PROGRAM P61_AO
VAR
	//ACT_Ramp_OLD();
	MFC01, MFC02, MFC03, MFC04, MFC05, MFC06, MFC07, MFC08, MFC09, MFC10: FB_Ramp2;
	MFC11, MFC12, MFC13, MFC14, MFC15, MFC16, MFC17, MFC18, MFC19: FB_Ramp2;		
	EPC01, EPC02, EPC03, EPC04, EPC05, EPC06, EPC07: FB_Ramp2;	
	IH, ROT, POS, P01: FB_Ramp2;
		
	//HT01: FB_Ramp2;
	halfRes: REAL := 16383;//0~5V
	fullRes: REAL := 32767;//0~10V or 4~20mA
	halfRes_ROT: REAL := 13106;//0~4V : 0 ~ 2500RPM - BLHM230K-GFS
		
	M01, M02, M03, M04, M05, M06, M07, M08, M09, M10: FB_Ramp_0;
	M11, M12, M13, M14, M15, M16, M17, M18, M19: FB_Ramp_0;	
	E01, E02, E03, E04, E05, E06, E07: FB_Ramp_0;	
	IH_0, ROT_0, POS_0, P01_0: FB_Ramp_0;
END_VAR

//IF EN_RUN_RCP = Off THEN
	ACT_Ramp();
//	ACT_Ramp_OLD();	
//END_IF

//----------------------------Analog Output--------------------------
IF N_MAX[0] > 0 THEN YA_M01 := REAL_TO_WORD(sv_M01 * halfRes / N_MAX[0]); END_IF;//MFC01 : 0~5V
IF N_MAX[1] > 0 THEN YA_M02 := REAL_TO_WORD(sv_M02 * halfRes / N_MAX[1]); END_IF;//MFC02 : 0~5V
IF N_MAX[2] > 0 THEN YA_M03 := REAL_TO_WORD(sv_M03 * halfRes / N_MAX[2]); END_IF;//MFC03 : 0~5V
IF N_MAX[3] > 0 THEN YA_M04 := REAL_TO_WORD(sv_M04 * halfRes / N_MAX[3]); END_IF;//MFC04 : 0~5V
IF N_MAX[4] > 0 THEN YA_M05 := REAL_TO_WORD(sv_M05 * halfRes / N_MAX[4]); END_IF;//MFC05 : 0~5V
IF N_MAX[5] > 0 THEN YA_M06 := REAL_TO_WORD(sv_M06 * halfRes / N_MAX[5]); END_IF;//MFC06 : 0~5V
IF N_MAX[6] > 0 THEN YA_M07 := REAL_TO_WORD(sv_M07 * halfRes / N_MAX[6]); END_IF;//MFC07 : 0~5V       
IF N_MAX[7] > 0 THEN YA_M08 := REAL_TO_WORD(sv_M08 * halfRes / N_MAX[7]); END_IF;//MFC08 : 0~5V
IF N_MAX[8] > 0 THEN YA_M09 := REAL_TO_WORD(sv_M09 * halfRes / N_MAX[8]); END_IF;//MFC09 : 0~5V
IF N_MAX[9] > 0 THEN YA_M10 := REAL_TO_WORD(sv_M10 * halfRes / N_MAX[9]); END_IF;//MFC10 : 0~5V
IF N_MAX[10] > 0 THEN YA_M11 := REAL_TO_WORD(sv_M11 * halfRes / N_MAX[10]); END_IF;//MFC11 : 0~5V
IF N_MAX[11] > 0 THEN YA_M12 := REAL_TO_WORD(sv_M12 * halfRes / N_MAX[11]); END_IF;//MFC12 : 0~5V
IF N_MAX[12] > 0 THEN YA_M13 := REAL_TO_WORD(sv_M13 * halfRes / N_MAX[12]); END_IF;//MFC13 : 0~5V
IF N_MAX[13] > 0 THEN YA_M14 := REAL_TO_WORD(sv_M14 * halfRes / N_MAX[13]); END_IF;//MFC14 : 0~5V
IF N_MAX[14] > 0 THEN YA_M15 := REAL_TO_WORD(sv_M15 * halfRes / N_MAX[14]); END_IF;//MFC15 : 0~5V
IF N_MAX[15] > 0 THEN YA_M16 := REAL_TO_WORD(sv_M16 * halfRes / N_MAX[15]); END_IF;//MFC16 : 0~5V
IF N_MAX[16] > 0 THEN YA_M17 := REAL_TO_WORD(sv_M17 * halfRes / N_MAX[16]); END_IF;//MFC17 : 0~5V
IF N_MAX[17] > 0 THEN YA_M18 := REAL_TO_WORD(sv_M18 * halfRes / N_MAX[17]); END_IF;//MFC18 : 0~5V
IF N_MAX[18] > 0 THEN YA_M19 := REAL_TO_WORD(sv_M19 * halfRes / N_MAX[18]); END_IF;//MFC19 : 0~5V
IF N_MAX[19] > 0 THEN YA_E01 := REAL_TO_WORD(sv_E01 * halfRes / N_MAX[19]); END_IF;//EPC01 : 0~5V
IF N_MAX[20] > 0 THEN YA_E02 := REAL_TO_WORD(sv_E02 * halfRes / N_MAX[20]); END_IF;//EPC02 : 0~5V
IF N_MAX[21] > 0 THEN YA_E03 := REAL_TO_WORD(sv_E03 * halfRes / N_MAX[21]); END_IF;//EPC03 : 0~5V
IF N_MAX[22] > 0 THEN YA_E04 := REAL_TO_WORD(sv_E04 * halfRes / N_MAX[22]); END_IF;//EPC04 : 0~5V
IF N_MAX[23] > 0 THEN YA_E05 := REAL_TO_WORD(sv_E05 * halfRes / N_MAX[23]); END_IF;//EPC05 : 0~5V
IF N_MAX[24] > 0 THEN YA_E06 := REAL_TO_WORD(sv_E06 * halfRes / N_MAX[24]); END_IF;//EPC06 : 0~5V
IF N_MAX[25] > 0 THEN YA_E07 := REAL_TO_WORD(sv_E07 * halfRes / N_MAX[25]); END_IF;//EPC07 : 0~5V
YA_P03 := XA_P03;//Exhaust Pressure(1000 Torr) Display-> AM215A-13  : 0~10V  
//IF N_MAX[26] > 0 THEN YA_Temp := REAL_TO_WORD(sv_IHT * fullRes / N_MAX[26]); END_IF;//IH - E3508 - DeviceNet
IF N_MAX[27] > 0 THEN YA_ROT := REAL_TO_WORD(e_ROT_AO_OFFSET + (sv_ROT * halfRes_ROT / N_MAX[27]) * e_ROT_AO_SLOPE_FACTOR); END_IF;//ROT : 0~4V
//IF N_MAX[27] > 0 THEN YA_ROT := REAL_TO_WORD(sv_ROT * halfRes_ROT / N_MAX[27]); END_IF;//ROT : 0~4V
//IF N_MAX[28] > 0 THEN YA_TV := REAL_TO_WORD(sv_TV * fullRes / N_MAX[28]); END_IF;//TV Position- Nocal - DeviceNet
//IF N_MAX[29] > 0 THEN YA_P01 := REAL_TO_WORD(sv_P01 * fullRes / N_MAX[29]); END_IF;//TV Pressure- Nocal - DeviceNet

ACTION ACT_Ramp:
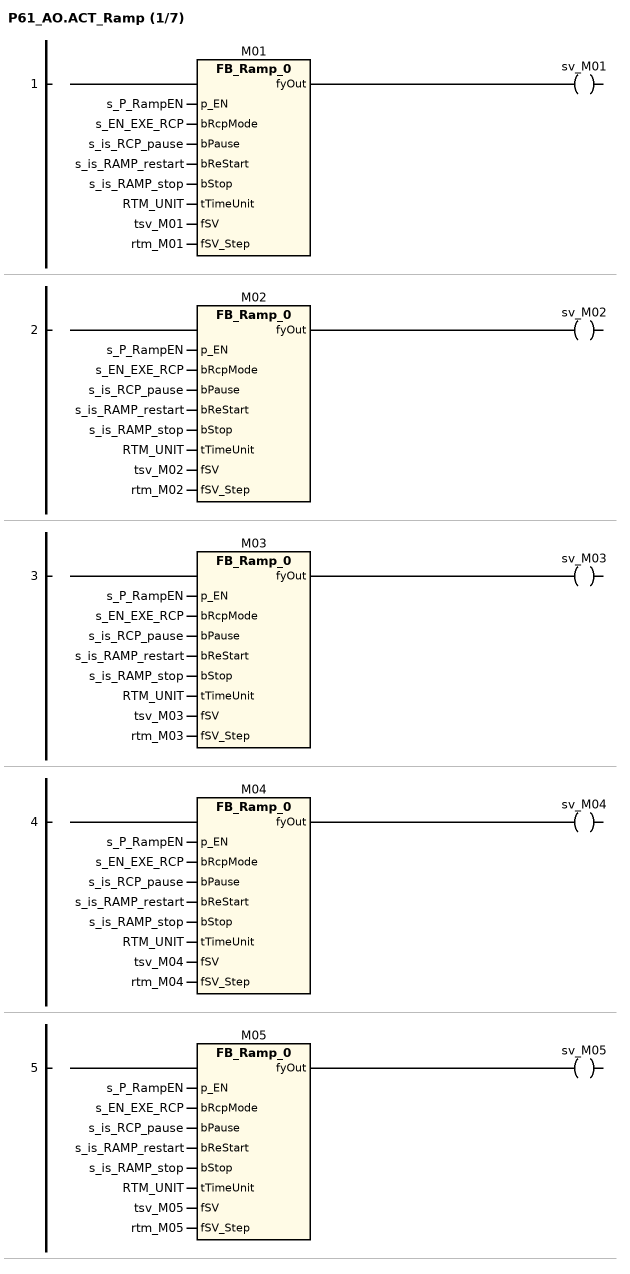
// NETWORK 1
M01(
    p_EN := s_P_RampEN,
    bRcpMode := s_EN_EXE_RCP,
    bPause := s_is_RCP_pause,
    bReStart := s_is_RAMP_restart,
    bStop := s_is_RAMP_stop,
    tTimeUnit := RTM_UNIT,
    fSV := tsv_M01,
    fSV_Step := rtm_M01); // FB_Ramp_0
sv_M01 := M01.fyOut;

// NETWORK 2
M02(
    p_EN := s_P_RampEN,
    bRcpMode := s_EN_EXE_RCP,
    bPause := s_is_RCP_pause,
    bReStart := s_is_RAMP_restart,
    bStop := s_is_RAMP_stop,
    tTimeUnit := RTM_UNIT,
    fSV := tsv_M02,
    fSV_Step := rtm_M02); // FB_Ramp_0
sv_M02 := M02.fyOut;

// NETWORK 3
M03(
    p_EN := s_P_RampEN,
    bRcpMode := s_EN_EXE_RCP,
    bPause := s_is_RCP_pause,
    bReStart := s_is_RAMP_restart,
    bStop := s_is_RAMP_stop,
    tTimeUnit := RTM_UNIT,
    fSV := tsv_M03,
    fSV_Step := rtm_M03); // FB_Ramp_0
sv_M03 := M03.fyOut;

// NETWORK 4
M04(
    p_EN := s_P_RampEN,
    bRcpMode := s_EN_EXE_RCP,
    bPause := s_is_RCP_pause,
    bReStart := s_is_RAMP_restart,
    bStop := s_is_RAMP_stop,
    tTimeUnit := RTM_UNIT,
    fSV := tsv_M04,
    fSV_Step := rtm_M04); // FB_Ramp_0
sv_M04 := M04.fyOut;

// NETWORK 5
M05(
    p_EN := s_P_RampEN,
    bRcpMode := s_EN_EXE_RCP,
    bPause := s_is_RCP_pause,
    bReStart := s_is_RAMP_restart,
    bStop := s_is_RAMP_stop,
    tTimeUnit := RTM_UNIT,
    fSV := tsv_M05,
    fSV_Step := rtm_M05); // FB_Ramp_0
sv_M05 := M05.fyOut;

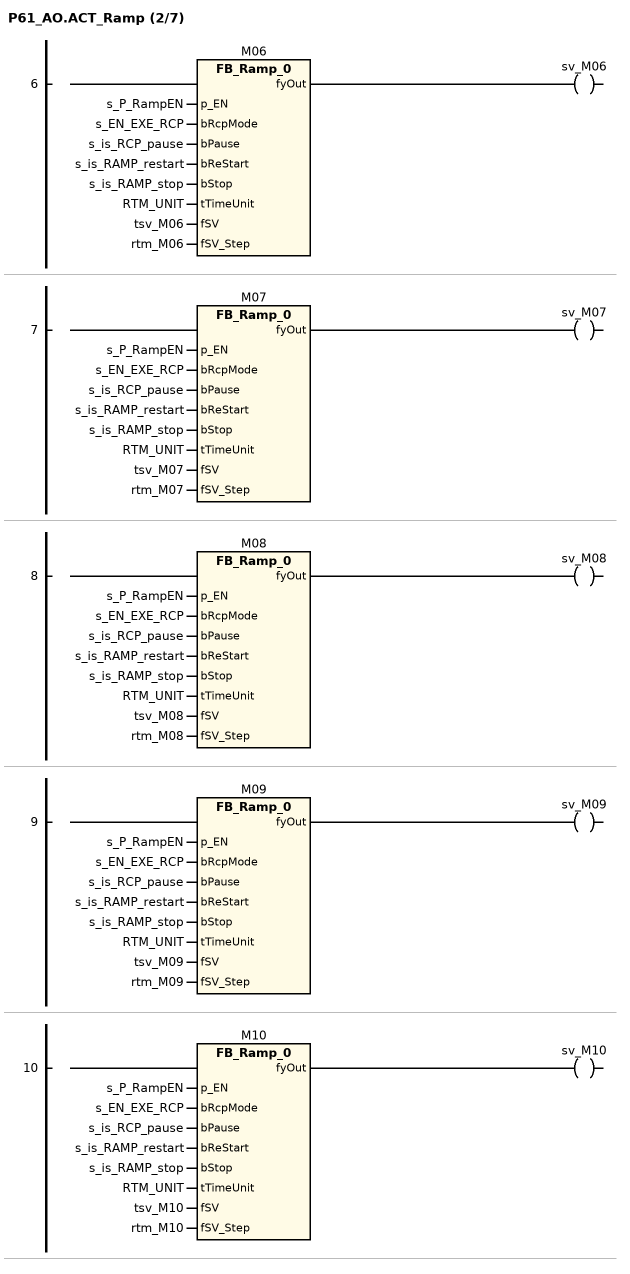
// NETWORK 6
M06(
    p_EN := s_P_RampEN,
    bRcpMode := s_EN_EXE_RCP,
    bPause := s_is_RCP_pause,
    bReStart := s_is_RAMP_restart,
    bStop := s_is_RAMP_stop,
    tTimeUnit := RTM_UNIT,
    fSV := tsv_M06,
    fSV_Step := rtm_M06); // FB_Ramp_0
sv_M06 := M06.fyOut;

// NETWORK 7
M07(
    p_EN := s_P_RampEN,
    bRcpMode := s_EN_EXE_RCP,
    bPause := s_is_RCP_pause,
    bReStart := s_is_RAMP_restart,
    bStop := s_is_RAMP_stop,
    tTimeUnit := RTM_UNIT,
    fSV := tsv_M07,
    fSV_Step := rtm_M07); // FB_Ramp_0
sv_M07 := M07.fyOut;

// NETWORK 8
M08(
    p_EN := s_P_RampEN,
    bRcpMode := s_EN_EXE_RCP,
    bPause := s_is_RCP_pause,
    bReStart := s_is_RAMP_restart,
    bStop := s_is_RAMP_stop,
    tTimeUnit := RTM_UNIT,
    fSV := tsv_M08,
    fSV_Step := rtm_M08); // FB_Ramp_0
sv_M08 := M08.fyOut;

// NETWORK 9
M09(
    p_EN := s_P_RampEN,
    bRcpMode := s_EN_EXE_RCP,
    bPause := s_is_RCP_pause,
    bReStart := s_is_RAMP_restart,
    bStop := s_is_RAMP_stop,
    tTimeUnit := RTM_UNIT,
    fSV := tsv_M09,
    fSV_Step := rtm_M09); // FB_Ramp_0
sv_M09 := M09.fyOut;

// NETWORK 10
M10(
    p_EN := s_P_RampEN,
    bRcpMode := s_EN_EXE_RCP,
    bPause := s_is_RCP_pause,
    bReStart := s_is_RAMP_restart,
    bStop := s_is_RAMP_stop,
    tTimeUnit := RTM_UNIT,
    fSV := tsv_M10,
    fSV_Step := rtm_M10); // FB_Ramp_0
sv_M10 := M10.fyOut;

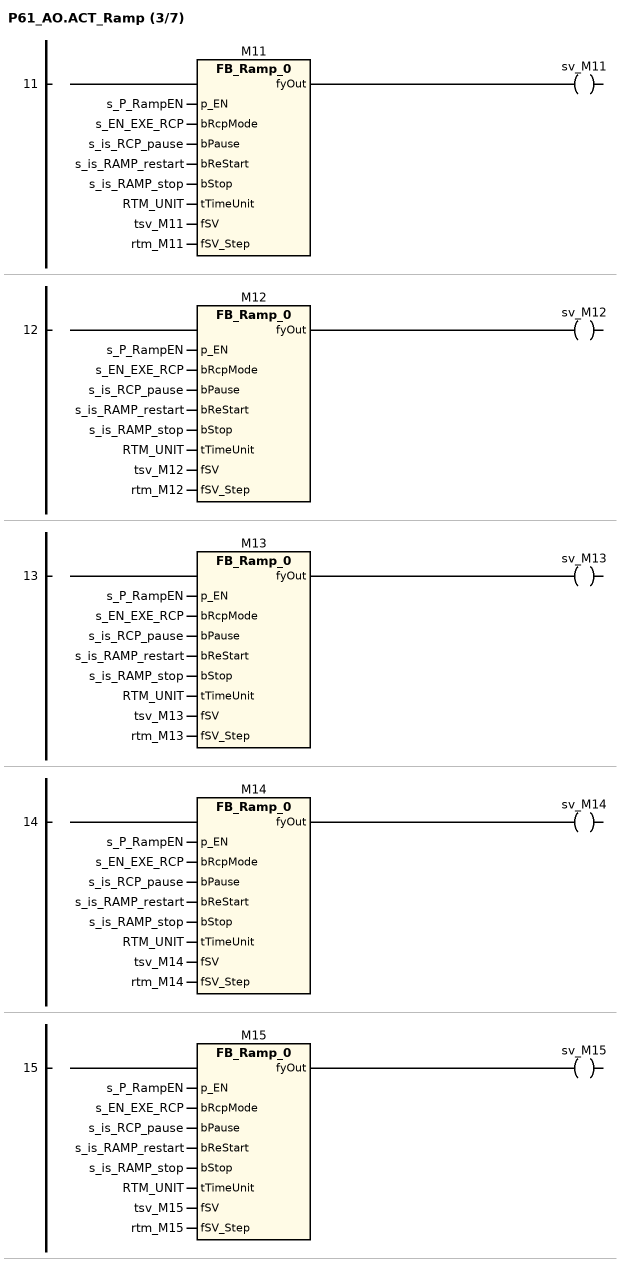
// NETWORK 11
M11(
    p_EN := s_P_RampEN,
    bRcpMode := s_EN_EXE_RCP,
    bPause := s_is_RCP_pause,
    bReStart := s_is_RAMP_restart,
    bStop := s_is_RAMP_stop,
    tTimeUnit := RTM_UNIT,
    fSV := tsv_M11,
    fSV_Step := rtm_M11); // FB_Ramp_0
sv_M11 := M11.fyOut;

// NETWORK 12
M12(
    p_EN := s_P_RampEN,
    bRcpMode := s_EN_EXE_RCP,
    bPause := s_is_RCP_pause,
    bReStart := s_is_RAMP_restart,
    bStop := s_is_RAMP_stop,
    tTimeUnit := RTM_UNIT,
    fSV := tsv_M12,
    fSV_Step := rtm_M12); // FB_Ramp_0
sv_M12 := M12.fyOut;

// NETWORK 13
M13(
    p_EN := s_P_RampEN,
    bRcpMode := s_EN_EXE_RCP,
    bPause := s_is_RCP_pause,
    bReStart := s_is_RAMP_restart,
    bStop := s_is_RAMP_stop,
    tTimeUnit := RTM_UNIT,
    fSV := tsv_M13,
    fSV_Step := rtm_M13); // FB_Ramp_0
sv_M13 := M13.fyOut;

// NETWORK 14
M14(
    p_EN := s_P_RampEN,
    bRcpMode := s_EN_EXE_RCP,
    bPause := s_is_RCP_pause,
    bReStart := s_is_RAMP_restart,
    bStop := s_is_RAMP_stop,
    tTimeUnit := RTM_UNIT,
    fSV := tsv_M14,
    fSV_Step := rtm_M14); // FB_Ramp_0
sv_M14 := M14.fyOut;

// NETWORK 15
M15(
    p_EN := s_P_RampEN,
    bRcpMode := s_EN_EXE_RCP,
    bPause := s_is_RCP_pause,
    bReStart := s_is_RAMP_restart,
    bStop := s_is_RAMP_stop,
    tTimeUnit := RTM_UNIT,
    fSV := tsv_M15,
    fSV_Step := rtm_M15); // FB_Ramp_0
sv_M15 := M15.fyOut;

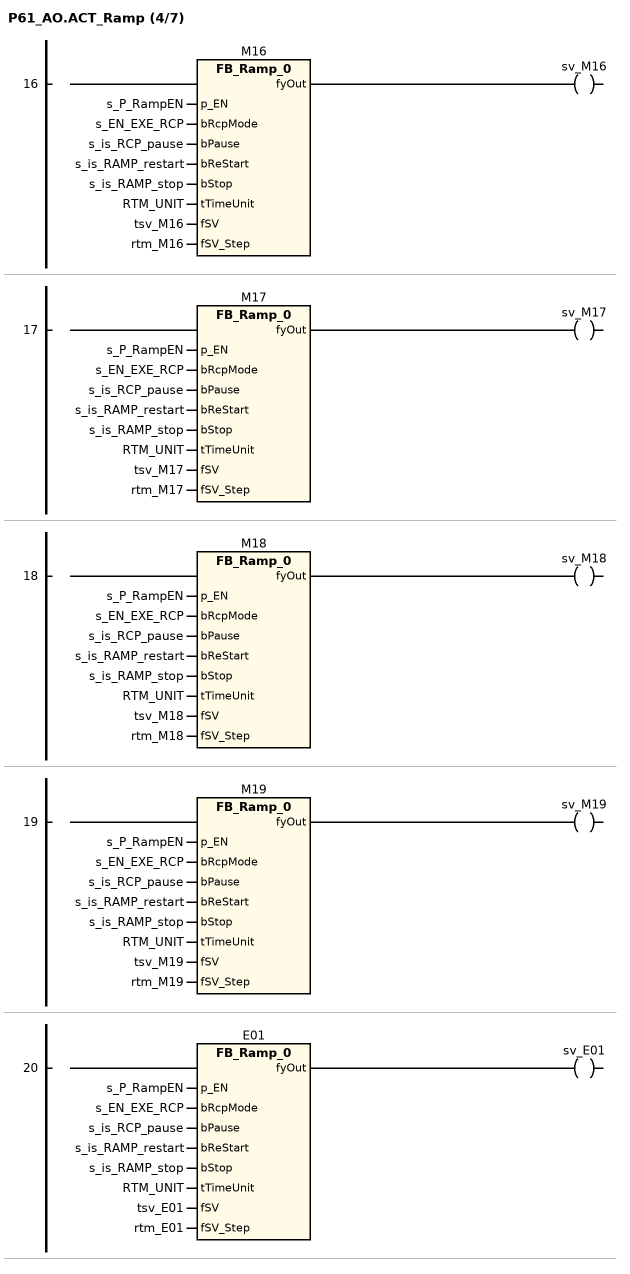
// NETWORK 16
M16(
    p_EN := s_P_RampEN,
    bRcpMode := s_EN_EXE_RCP,
    bPause := s_is_RCP_pause,
    bReStart := s_is_RAMP_restart,
    bStop := s_is_RAMP_stop,
    tTimeUnit := RTM_UNIT,
    fSV := tsv_M16,
    fSV_Step := rtm_M16); // FB_Ramp_0
sv_M16 := M16.fyOut;

// NETWORK 17
M17(
    p_EN := s_P_RampEN,
    bRcpMode := s_EN_EXE_RCP,
    bPause := s_is_RCP_pause,
    bReStart := s_is_RAMP_restart,
    bStop := s_is_RAMP_stop,
    tTimeUnit := RTM_UNIT,
    fSV := tsv_M17,
    fSV_Step := rtm_M17); // FB_Ramp_0
sv_M17 := M17.fyOut;

// NETWORK 18
M18(
    p_EN := s_P_RampEN,
    bRcpMode := s_EN_EXE_RCP,
    bPause := s_is_RCP_pause,
    bReStart := s_is_RAMP_restart,
    bStop := s_is_RAMP_stop,
    tTimeUnit := RTM_UNIT,
    fSV := tsv_M18,
    fSV_Step := rtm_M18); // FB_Ramp_0
sv_M18 := M18.fyOut;

// NETWORK 19
M19(
    p_EN := s_P_RampEN,
    bRcpMode := s_EN_EXE_RCP,
    bPause := s_is_RCP_pause,
    bReStart := s_is_RAMP_restart,
    bStop := s_is_RAMP_stop,
    tTimeUnit := RTM_UNIT,
    fSV := tsv_M19,
    fSV_Step := rtm_M19); // FB_Ramp_0
sv_M19 := M19.fyOut;

// NETWORK 20
E01(
    p_EN := s_P_RampEN,
    bRcpMode := s_EN_EXE_RCP,
    bPause := s_is_RCP_pause,
    bReStart := s_is_RAMP_restart,
    bStop := s_is_RAMP_stop,
    tTimeUnit := RTM_UNIT,
    fSV := tsv_E01,
    fSV_Step := rtm_E01); // FB_Ramp_0
sv_E01 := E01.fyOut;

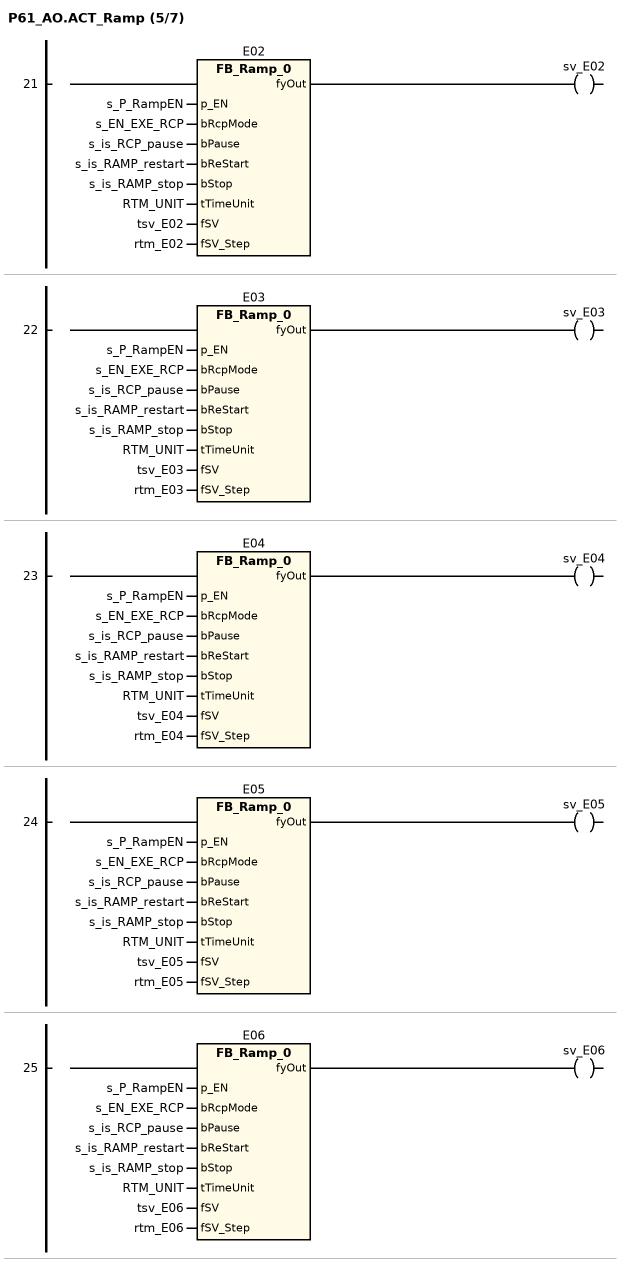
// NETWORK 21
E02(
    p_EN := s_P_RampEN,
    bRcpMode := s_EN_EXE_RCP,
    bPause := s_is_RCP_pause,
    bReStart := s_is_RAMP_restart,
    bStop := s_is_RAMP_stop,
    tTimeUnit := RTM_UNIT,
    fSV := tsv_E02,
    fSV_Step := rtm_E02); // FB_Ramp_0
sv_E02 := E02.fyOut;

// NETWORK 22
E03(
    p_EN := s_P_RampEN,
    bRcpMode := s_EN_EXE_RCP,
    bPause := s_is_RCP_pause,
    bReStart := s_is_RAMP_restart,
    bStop := s_is_RAMP_stop,
    tTimeUnit := RTM_UNIT,
    fSV := tsv_E03,
    fSV_Step := rtm_E03); // FB_Ramp_0
sv_E03 := E03.fyOut;

// NETWORK 23
E04(
    p_EN := s_P_RampEN,
    bRcpMode := s_EN_EXE_RCP,
    bPause := s_is_RCP_pause,
    bReStart := s_is_RAMP_restart,
    bStop := s_is_RAMP_stop,
    tTimeUnit := RTM_UNIT,
    fSV := tsv_E04,
    fSV_Step := rtm_E04); // FB_Ramp_0
sv_E04 := E04.fyOut;

// NETWORK 24
E05(
    p_EN := s_P_RampEN,
    bRcpMode := s_EN_EXE_RCP,
    bPause := s_is_RCP_pause,
    bReStart := s_is_RAMP_restart,
    bStop := s_is_RAMP_stop,
    tTimeUnit := RTM_UNIT,
    fSV := tsv_E05,
    fSV_Step := rtm_E05); // FB_Ramp_0
sv_E05 := E05.fyOut;

// NETWORK 25
E06(
    p_EN := s_P_RampEN,
    bRcpMode := s_EN_EXE_RCP,
    bPause := s_is_RCP_pause,
    bReStart := s_is_RAMP_restart,
    bStop := s_is_RAMP_stop,
    tTimeUnit := RTM_UNIT,
    fSV := tsv_E06,
    fSV_Step := rtm_E06); // FB_Ramp_0
sv_E06 := E06.fyOut;

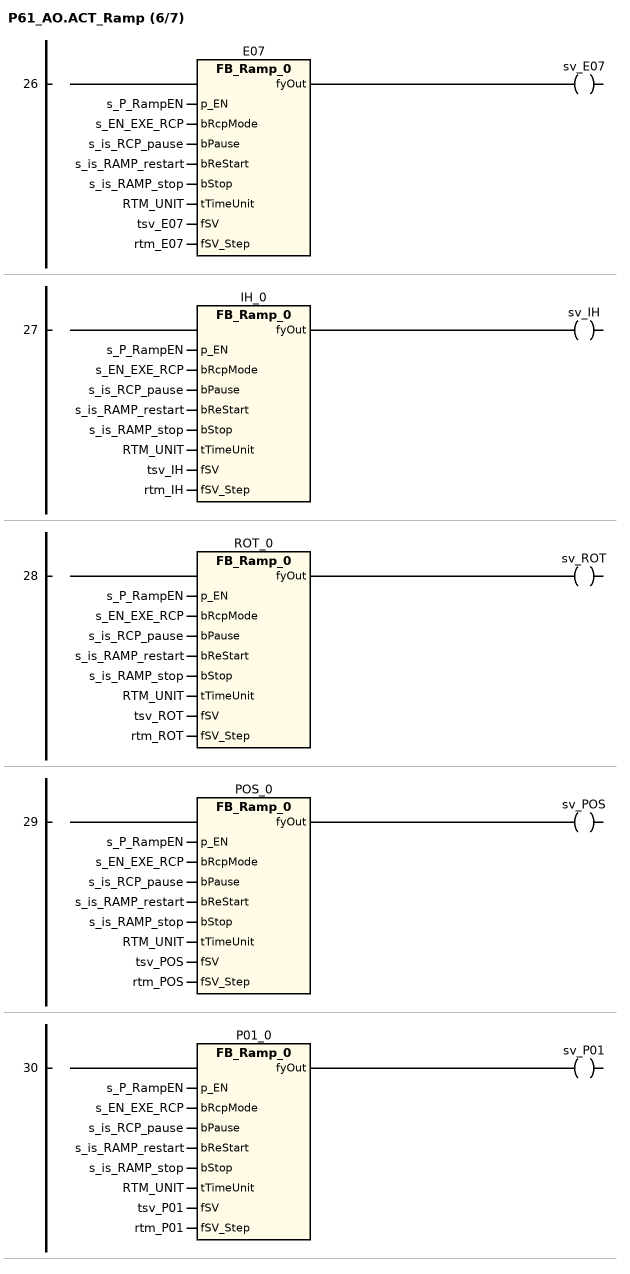
// NETWORK 26
E07(
    p_EN := s_P_RampEN,
    bRcpMode := s_EN_EXE_RCP,
    bPause := s_is_RCP_pause,
    bReStart := s_is_RAMP_restart,
    bStop := s_is_RAMP_stop,
    tTimeUnit := RTM_UNIT,
    fSV := tsv_E07,
    fSV_Step := rtm_E07); // FB_Ramp_0
sv_E07 := E07.fyOut;

// NETWORK 27
IH_0(
    p_EN := s_P_RampEN,
    bRcpMode := s_EN_EXE_RCP,
    bPause := s_is_RCP_pause,
    bReStart := s_is_RAMP_restart,
    bStop := s_is_RAMP_stop,
    tTimeUnit := RTM_UNIT,
    fSV := tsv_IH,
    fSV_Step := rtm_IH); // FB_Ramp_0
sv_IH := IH_0.fyOut;

// NETWORK 28
ROT_0(
    p_EN := s_P_RampEN,
    bRcpMode := s_EN_EXE_RCP,
    bPause := s_is_RCP_pause,
    bReStart := s_is_RAMP_restart,
    bStop := s_is_RAMP_stop,
    tTimeUnit := RTM_UNIT,
    fSV := tsv_ROT,
    fSV_Step := rtm_ROT); // FB_Ramp_0
sv_ROT := ROT_0.fyOut;

// NETWORK 29
POS_0(
    p_EN := s_P_RampEN,
    bRcpMode := s_EN_EXE_RCP,
    bPause := s_is_RCP_pause,
    bReStart := s_is_RAMP_restart,
    bStop := s_is_RAMP_stop,
    tTimeUnit := RTM_UNIT,
    fSV := tsv_POS,
    fSV_Step := rtm_POS); // FB_Ramp_0
sv_POS := POS_0.fyOut;

// NETWORK 30
P01_0(
    p_EN := s_P_RampEN,
    bRcpMode := s_EN_EXE_RCP,
    bPause := s_is_RCP_pause,
    bReStart := s_is_RAMP_restart,
    bStop := s_is_RAMP_stop,
    tTimeUnit := RTM_UNIT,
    fSV := tsv_P01,
    fSV_Step := rtm_P01); // FB_Ramp_0
sv_P01 := P01_0.fyOut;

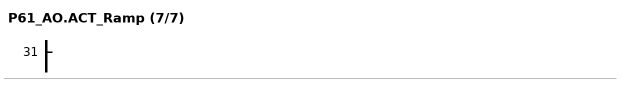
// NETWORK 31
END_ACTION

ACTION ACT_Ramp_OLD:
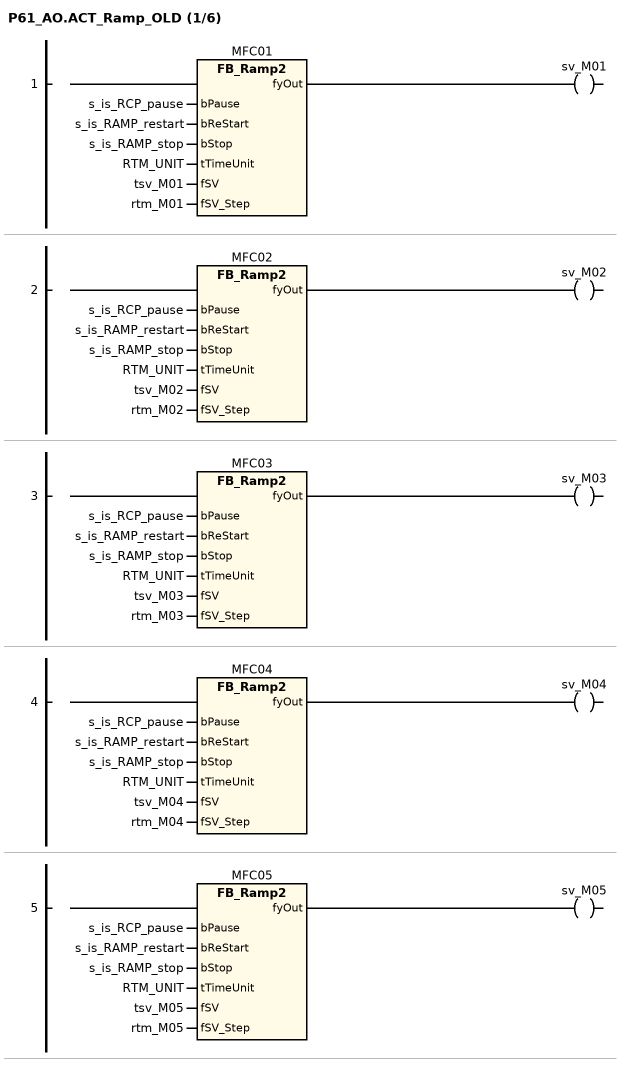
// NETWORK 1
MFC01(
    bPause := s_is_RCP_pause,
    bReStart := s_is_RAMP_restart,
    bStop := s_is_RAMP_stop,
    tTimeUnit := RTM_UNIT,
    fSV := tsv_M01,
    fSV_Step := rtm_M01); // FB_Ramp2
sv_M01 := MFC01.fyOut;

// NETWORK 2
MFC02(
    bPause := s_is_RCP_pause,
    bReStart := s_is_RAMP_restart,
    bStop := s_is_RAMP_stop,
    tTimeUnit := RTM_UNIT,
    fSV := tsv_M02,
    fSV_Step := rtm_M02); // FB_Ramp2
sv_M02 := MFC02.fyOut;

// NETWORK 3
MFC03(
    bPause := s_is_RCP_pause,
    bReStart := s_is_RAMP_restart,
    bStop := s_is_RAMP_stop,
    tTimeUnit := RTM_UNIT,
    fSV := tsv_M03,
    fSV_Step := rtm_M03); // FB_Ramp2
sv_M03 := MFC03.fyOut;

// NETWORK 4
MFC04(
    bPause := s_is_RCP_pause,
    bReStart := s_is_RAMP_restart,
    bStop := s_is_RAMP_stop,
    tTimeUnit := RTM_UNIT,
    fSV := tsv_M04,
    fSV_Step := rtm_M04); // FB_Ramp2
sv_M04 := MFC04.fyOut;

// NETWORK 5
MFC05(
    bPause := s_is_RCP_pause,
    bReStart := s_is_RAMP_restart,
    bStop := s_is_RAMP_stop,
    tTimeUnit := RTM_UNIT,
    fSV := tsv_M05,
    fSV_Step := rtm_M05); // FB_Ramp2
sv_M05 := MFC05.fyOut;

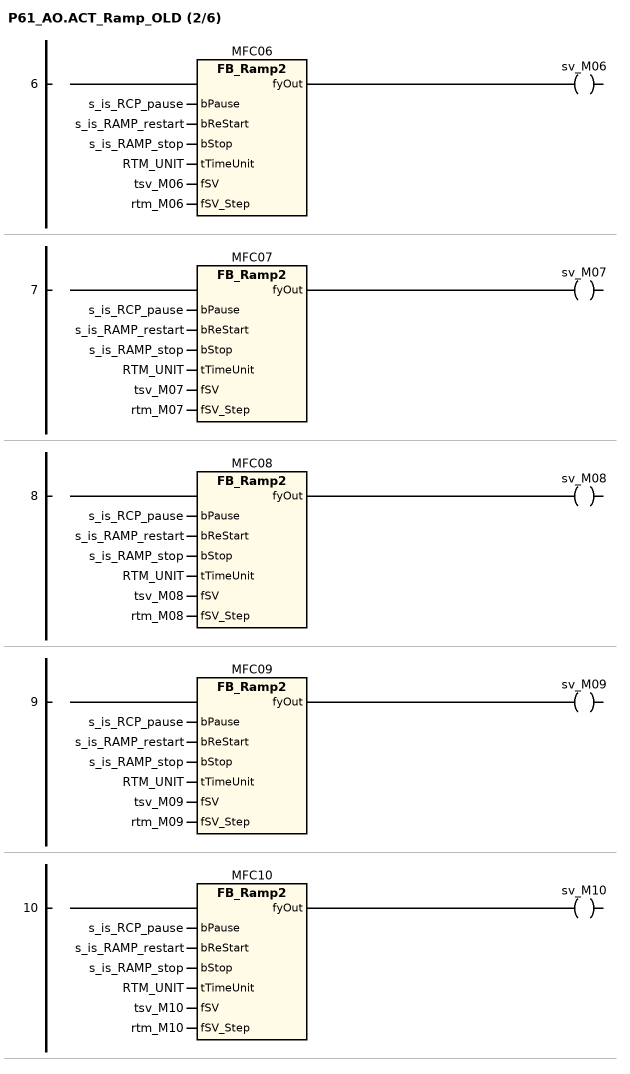
// NETWORK 6
MFC06(
    bPause := s_is_RCP_pause,
    bReStart := s_is_RAMP_restart,
    bStop := s_is_RAMP_stop,
    tTimeUnit := RTM_UNIT,
    fSV := tsv_M06,
    fSV_Step := rtm_M06); // FB_Ramp2
sv_M06 := MFC06.fyOut;

// NETWORK 7
MFC07(
    bPause := s_is_RCP_pause,
    bReStart := s_is_RAMP_restart,
    bStop := s_is_RAMP_stop,
    tTimeUnit := RTM_UNIT,
    fSV := tsv_M07,
    fSV_Step := rtm_M07); // FB_Ramp2
sv_M07 := MFC07.fyOut;

// NETWORK 8
MFC08(
    bPause := s_is_RCP_pause,
    bReStart := s_is_RAMP_restart,
    bStop := s_is_RAMP_stop,
    tTimeUnit := RTM_UNIT,
    fSV := tsv_M08,
    fSV_Step := rtm_M08); // FB_Ramp2
sv_M08 := MFC08.fyOut;

// NETWORK 9
MFC09(
    bPause := s_is_RCP_pause,
    bReStart := s_is_RAMP_restart,
    bStop := s_is_RAMP_stop,
    tTimeUnit := RTM_UNIT,
    fSV := tsv_M09,
    fSV_Step := rtm_M09); // FB_Ramp2
sv_M09 := MFC09.fyOut;

// NETWORK 10
MFC10(
    bPause := s_is_RCP_pause,
    bReStart := s_is_RAMP_restart,
    bStop := s_is_RAMP_stop,
    tTimeUnit := RTM_UNIT,
    fSV := tsv_M10,
    fSV_Step := rtm_M10); // FB_Ramp2
sv_M10 := MFC10.fyOut;

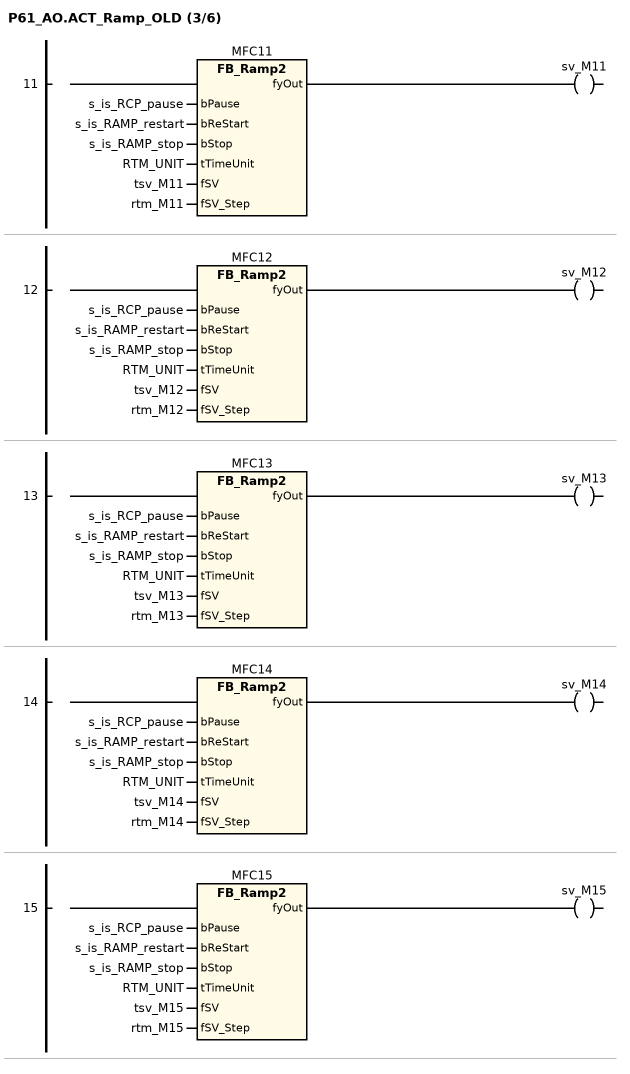
// NETWORK 11
MFC11(
    bPause := s_is_RCP_pause,
    bReStart := s_is_RAMP_restart,
    bStop := s_is_RAMP_stop,
    tTimeUnit := RTM_UNIT,
    fSV := tsv_M11,
    fSV_Step := rtm_M11); // FB_Ramp2
sv_M11 := MFC11.fyOut;

// NETWORK 12
MFC12(
    bPause := s_is_RCP_pause,
    bReStart := s_is_RAMP_restart,
    bStop := s_is_RAMP_stop,
    tTimeUnit := RTM_UNIT,
    fSV := tsv_M12,
    fSV_Step := rtm_M12); // FB_Ramp2
sv_M12 := MFC12.fyOut;

// NETWORK 13
MFC13(
    bPause := s_is_RCP_pause,
    bReStart := s_is_RAMP_restart,
    bStop := s_is_RAMP_stop,
    tTimeUnit := RTM_UNIT,
    fSV := tsv_M13,
    fSV_Step := rtm_M13); // FB_Ramp2
sv_M13 := MFC13.fyOut;

// NETWORK 14
MFC14(
    bPause := s_is_RCP_pause,
    bReStart := s_is_RAMP_restart,
    bStop := s_is_RAMP_stop,
    tTimeUnit := RTM_UNIT,
    fSV := tsv_M14,
    fSV_Step := rtm_M14); // FB_Ramp2
sv_M14 := MFC14.fyOut;

// NETWORK 15
MFC15(
    bPause := s_is_RCP_pause,
    bReStart := s_is_RAMP_restart,
    bStop := s_is_RAMP_stop,
    tTimeUnit := RTM_UNIT,
    fSV := tsv_M15,
    fSV_Step := rtm_M15); // FB_Ramp2
sv_M15 := MFC15.fyOut;

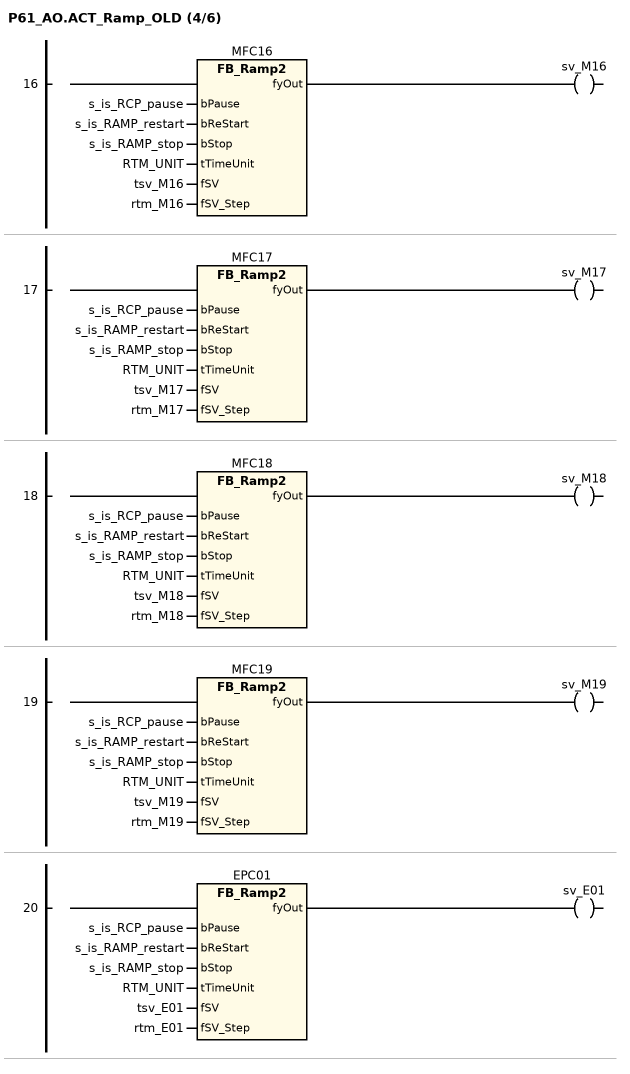
// NETWORK 16
MFC16(
    bPause := s_is_RCP_pause,
    bReStart := s_is_RAMP_restart,
    bStop := s_is_RAMP_stop,
    tTimeUnit := RTM_UNIT,
    fSV := tsv_M16,
    fSV_Step := rtm_M16); // FB_Ramp2
sv_M16 := MFC16.fyOut;

// NETWORK 17
MFC17(
    bPause := s_is_RCP_pause,
    bReStart := s_is_RAMP_restart,
    bStop := s_is_RAMP_stop,
    tTimeUnit := RTM_UNIT,
    fSV := tsv_M17,
    fSV_Step := rtm_M17); // FB_Ramp2
sv_M17 := MFC17.fyOut;

// NETWORK 18
MFC18(
    bPause := s_is_RCP_pause,
    bReStart := s_is_RAMP_restart,
    bStop := s_is_RAMP_stop,
    tTimeUnit := RTM_UNIT,
    fSV := tsv_M18,
    fSV_Step := rtm_M18); // FB_Ramp2
sv_M18 := MFC18.fyOut;

// NETWORK 19
MFC19(
    bPause := s_is_RCP_pause,
    bReStart := s_is_RAMP_restart,
    bStop := s_is_RAMP_stop,
    tTimeUnit := RTM_UNIT,
    fSV := tsv_M19,
    fSV_Step := rtm_M19); // FB_Ramp2
sv_M19 := MFC19.fyOut;

// NETWORK 20
EPC01(
    bPause := s_is_RCP_pause,
    bReStart := s_is_RAMP_restart,
    bStop := s_is_RAMP_stop,
    tTimeUnit := RTM_UNIT,
    fSV := tsv_E01,
    fSV_Step := rtm_E01); // FB_Ramp2
sv_E01 := EPC01.fyOut;

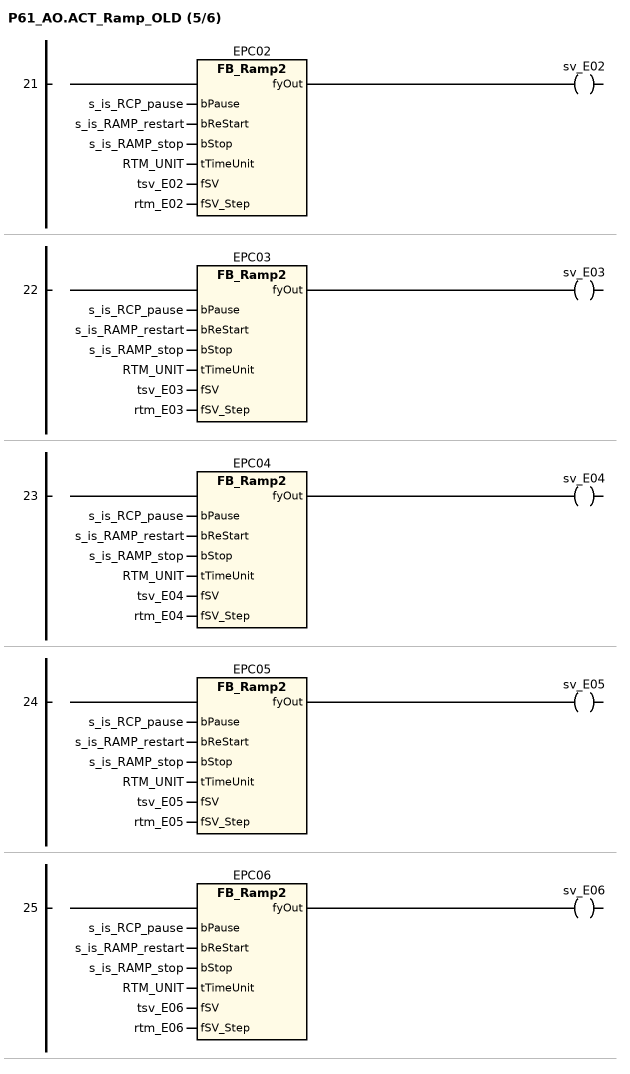
// NETWORK 21
EPC02(
    bPause := s_is_RCP_pause,
    bReStart := s_is_RAMP_restart,
    bStop := s_is_RAMP_stop,
    tTimeUnit := RTM_UNIT,
    fSV := tsv_E02,
    fSV_Step := rtm_E02); // FB_Ramp2
sv_E02 := EPC02.fyOut;

// NETWORK 22
EPC03(
    bPause := s_is_RCP_pause,
    bReStart := s_is_RAMP_restart,
    bStop := s_is_RAMP_stop,
    tTimeUnit := RTM_UNIT,
    fSV := tsv_E03,
    fSV_Step := rtm_E03); // FB_Ramp2
sv_E03 := EPC03.fyOut;

// NETWORK 23
EPC04(
    bPause := s_is_RCP_pause,
    bReStart := s_is_RAMP_restart,
    bStop := s_is_RAMP_stop,
    tTimeUnit := RTM_UNIT,
    fSV := tsv_E04,
    fSV_Step := rtm_E04); // FB_Ramp2
sv_E04 := EPC04.fyOut;

// NETWORK 24
EPC05(
    bPause := s_is_RCP_pause,
    bReStart := s_is_RAMP_restart,
    bStop := s_is_RAMP_stop,
    tTimeUnit := RTM_UNIT,
    fSV := tsv_E05,
    fSV_Step := rtm_E05); // FB_Ramp2
sv_E05 := EPC05.fyOut;

// NETWORK 25
EPC06(
    bPause := s_is_RCP_pause,
    bReStart := s_is_RAMP_restart,
    bStop := s_is_RAMP_stop,
    tTimeUnit := RTM_UNIT,
    fSV := tsv_E06,
    fSV_Step := rtm_E06); // FB_Ramp2
sv_E06 := EPC06.fyOut;

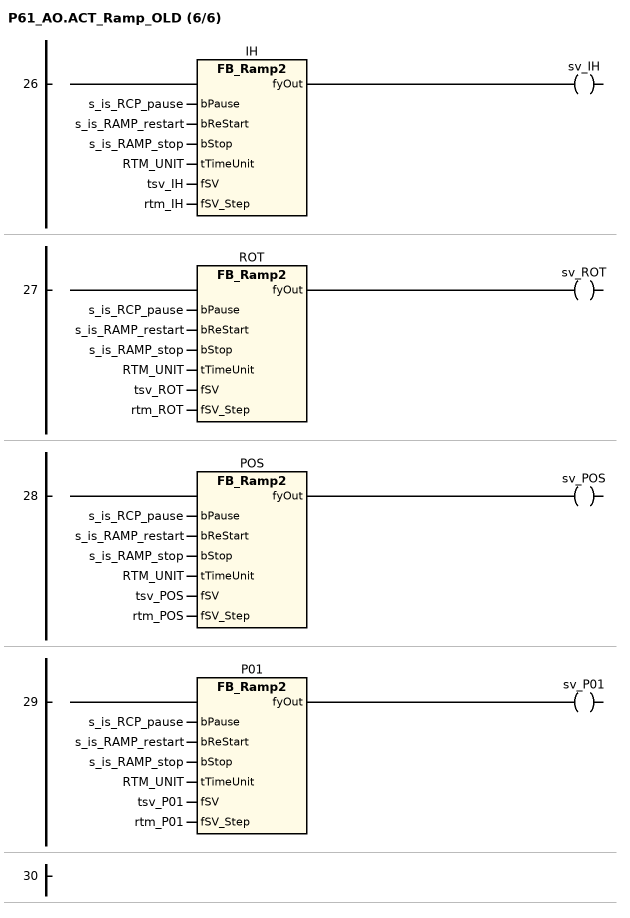
// NETWORK 26
IH(
    bPause := s_is_RCP_pause,
    bReStart := s_is_RAMP_restart,
    bStop := s_is_RAMP_stop,
    tTimeUnit := RTM_UNIT,
    fSV := tsv_IH,
    fSV_Step := rtm_IH); // FB_Ramp2
sv_IH := IH.fyOut;

// NETWORK 27
ROT(
    bPause := s_is_RCP_pause,
    bReStart := s_is_RAMP_restart,
    bStop := s_is_RAMP_stop,
    tTimeUnit := RTM_UNIT,
    fSV := tsv_ROT,
    fSV_Step := rtm_ROT); // FB_Ramp2
sv_ROT := ROT.fyOut;

// NETWORK 28
POS(
    bPause := s_is_RCP_pause,
    bReStart := s_is_RAMP_restart,
    bStop := s_is_RAMP_stop,
    tTimeUnit := RTM_UNIT,
    fSV := tsv_POS,
    fSV_Step := rtm_POS); // FB_Ramp2
sv_POS := POS.fyOut;

// NETWORK 29
P01(
    bPause := s_is_RCP_pause,
    bReStart := s_is_RAMP_restart,
    bStop := s_is_RAMP_stop,
    tTimeUnit := RTM_UNIT,
    fSV := tsv_P01,
    fSV_Step := rtm_P01); // FB_Ramp2
sv_P01 := P01.fyOut;

// NETWORK 30
END_ACTION

END_PROGRAM

(* stored: Version 1.1.0.1, ProductVersion 3.1.4024.12
   POU P61_AO: Id {aedf5e2e-3f2f-46cb-815a-6bb49535b436}, SpecialFunc None
   Action ACT_Ramp: Id {04785566-9696-4f5a-8d21-3829d3af1e91}
   Action ACT_Ramp_OLD: Id {f85f0e3a-0756-4081-b076-553964a3c377} *)
